// TIA Portal V17 export
// export: Created 2023-04-03T06:31:34.8487643Z, ExportSetting WithDefaults, DisplayName Totally Integrated Automation Portal, DisplayVersion V17 Update 4, DisplayName TIA Portal Openness, DisplayVersion V17 Update 4, DisplayName TIA Portal Version Control Interface, DisplayVersion V17, DisplayName STEP 7 Professional, DisplayVersion V17 Update 4, DisplayName STEP 7 Safety, DisplayVersion V17, DisplayName WinCC Professional, DisplayVersion V17 Update 4
FUNCTION "SM1_Logic" : Void   // FC60, LAD
TITLE = State Machine Logic
{ S7_Optimized_Access := 'TRUE' }
VERSION : 0.1
// stored: AutoNumber false, IsIECCheckEnabled false, SetENOAutomatically false, UDAEnableTagReadback false
   VAR_TEMP
      xStopSubSystem : Bool;
   END_VAR
   VAR_TEMP   // added for the SCL form of the ladder/FBD networks
      _w1 : Bool;
   END_VAR
BEGIN

REGION Network 1: Stop Command Local Mode
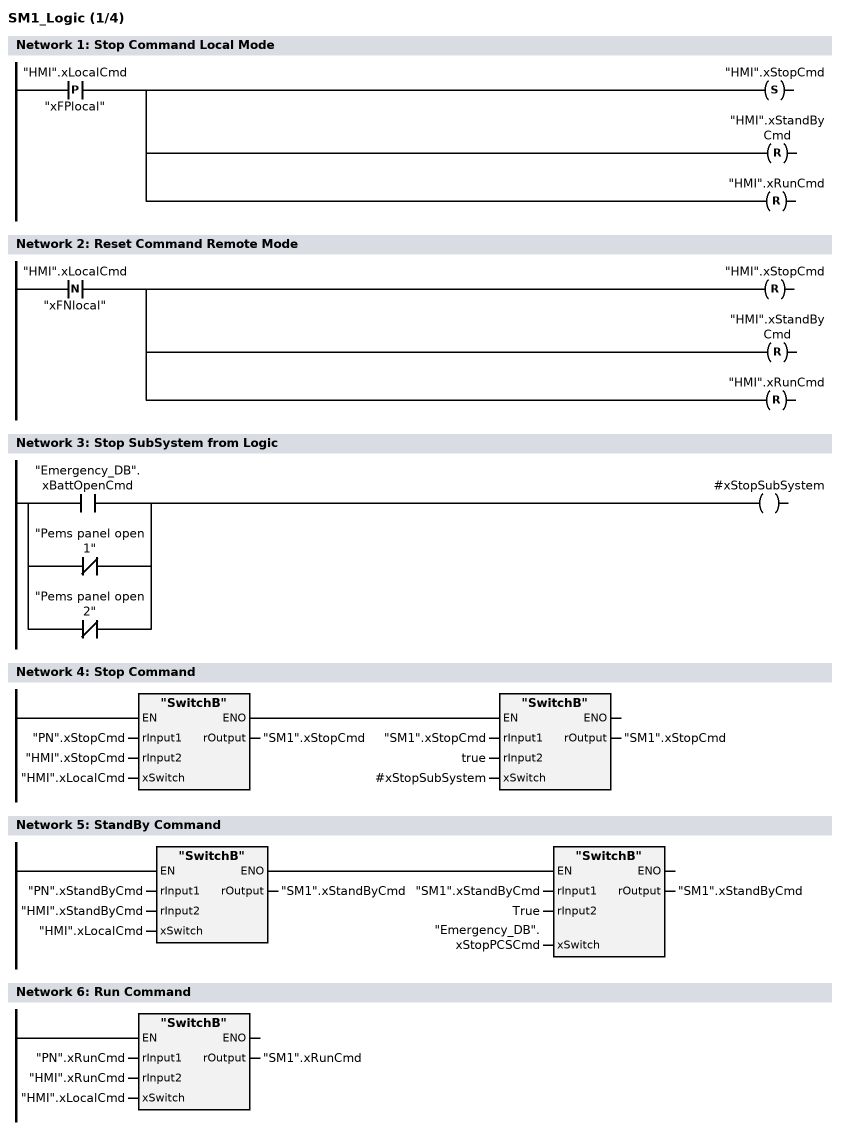
   RUNG wire#powerrail
      P_Contact(operand := "HMI".xLocalCmd, bit := "xFPlocal")
      wire#w1
      S_Coil( "HMI".xStopCmd )
   END_RUNG
   RUNG wire#w1
      R_Coil( "HMI".xStandByCmd )
   END_RUNG
   RUNG wire#w1
      R_Coil( "HMI".xRunCmd )
   END_RUNG
   // the same network as SCL:
   #_w1 := "HMI".xLocalCmd AND NOT "xFPlocal";   // rising edge of "HMI".xLocalCmd
   "xFPlocal" := "HMI".xLocalCmd;
   IF #_w1 THEN
       "HMI".xStopCmd := TRUE;
       "HMI".xStandByCmd := FALSE;
       "HMI".xRunCmd := FALSE;
   END_IF;
END_REGION

REGION Network 2: Reset Command Remote Mode
   RUNG wire#powerrail
      N_Contact(operand := "HMI".xLocalCmd, bit := "xFNlocal")
      wire#w1
      R_Coil( "HMI".xStopCmd )
   END_RUNG
   RUNG wire#w1
      R_Coil( "HMI".xStandByCmd )
   END_RUNG
   RUNG wire#w1
      R_Coil( "HMI".xRunCmd )
   END_RUNG
   // the same network as SCL:
   #_w1 := NOT "HMI".xLocalCmd AND "xFNlocal";   // falling edge of "HMI".xLocalCmd
   "xFNlocal" := "HMI".xLocalCmd;
   IF #_w1 THEN
       "HMI".xStopCmd := FALSE;
       "HMI".xStandByCmd := FALSE;
       "HMI".xRunCmd := FALSE;
   END_IF;
END_REGION

REGION Network 3: Stop SubSystem from Logic
   RUNG wire#powerrail
      Contact( "Emergency_DB".xBattOpenCmd )
      wire#w1
      Coil( #xStopSubSystem )
   END_RUNG
   RUNG wire#powerrail
      I_Contact( "Pems panel open 1" )
   END_RUNG wire#w1
   RUNG wire#powerrail
      I_Contact( "Pems panel open 2" )
   END_RUNG wire#w1
   // the same network as SCL:
   #xStopSubSystem := "Emergency_DB".xBattOpenCmd OR NOT "Pems panel open 1" OR NOT "Pems panel open 2";
END_REGION

REGION Network 4: Stop Command
   RUNG wire#powerrail
      "SwitchB"(rInput1 := "PN".xStopCmd, rInput2 := "HMI".xStopCmd, xSwitch := "HMI".xLocalCmd, rOutput => "SM1".xStopCmd)
      "SwitchB"(rInput1 := "SM1".xStopCmd, rInput2 := true, xSwitch := #xStopSubSystem, rOutput => "SM1".xStopCmd)
   END_RUNG
   // the same network as SCL:
   "SwitchB"(rInput1 := "PN".xStopCmd,
             rInput2 := "HMI".xStopCmd,
             xSwitch := "HMI".xLocalCmd,
             rOutput => "SM1".xStopCmd,
             ENO => #_w1);
   IF #_w1 THEN
       "SwitchB"(rInput1 := "SM1".xStopCmd, rInput2 := true, xSwitch := #xStopSubSystem, rOutput => "SM1".xStopCmd);
   END_IF;
END_REGION

REGION Network 5: StandBy Command
   RUNG wire#powerrail
      "SwitchB"(rInput1 := "PN".xStandByCmd, rInput2 := "HMI".xStandByCmd, xSwitch := "HMI".xLocalCmd, rOutput => "SM1".xStandByCmd)
      "SwitchB"(rInput1 := "SM1".xStandByCmd, rInput2 := True, xSwitch := "Emergency_DB".xStopPCSCmd, rOutput => "SM1".xStandByCmd)
   END_RUNG
   // the same network as SCL:
   "SwitchB"(rInput1 := "PN".xStandByCmd,
             rInput2 := "HMI".xStandByCmd,
             xSwitch := "HMI".xLocalCmd,
             rOutput => "SM1".xStandByCmd,
             ENO => #_w1);
   IF #_w1 THEN
       "SwitchB"(rInput1 := "SM1".xStandByCmd,
                 rInput2 := True,
                 xSwitch := "Emergency_DB".xStopPCSCmd,
                 rOutput => "SM1".xStandByCmd);
   END_IF;
END_REGION

REGION Network 6: Run Command
   RUNG wire#powerrail
      "SwitchB"(rInput1 := "PN".xRunCmd, rInput2 := "HMI".xRunCmd, xSwitch := "HMI".xLocalCmd, rOutput => "SM1".xRunCmd)
   END_RUNG
   // the same network as SCL:
   "SwitchB"(rInput1 := "PN".xRunCmd,
             rInput2 := "HMI".xRunCmd,
             xSwitch := "HMI".xLocalCmd,
             rOutput => "SM1".xRunCmd);
END_REGION

REGION Network 7: Local - Stop - StandBy - Run Status -> to HMI status
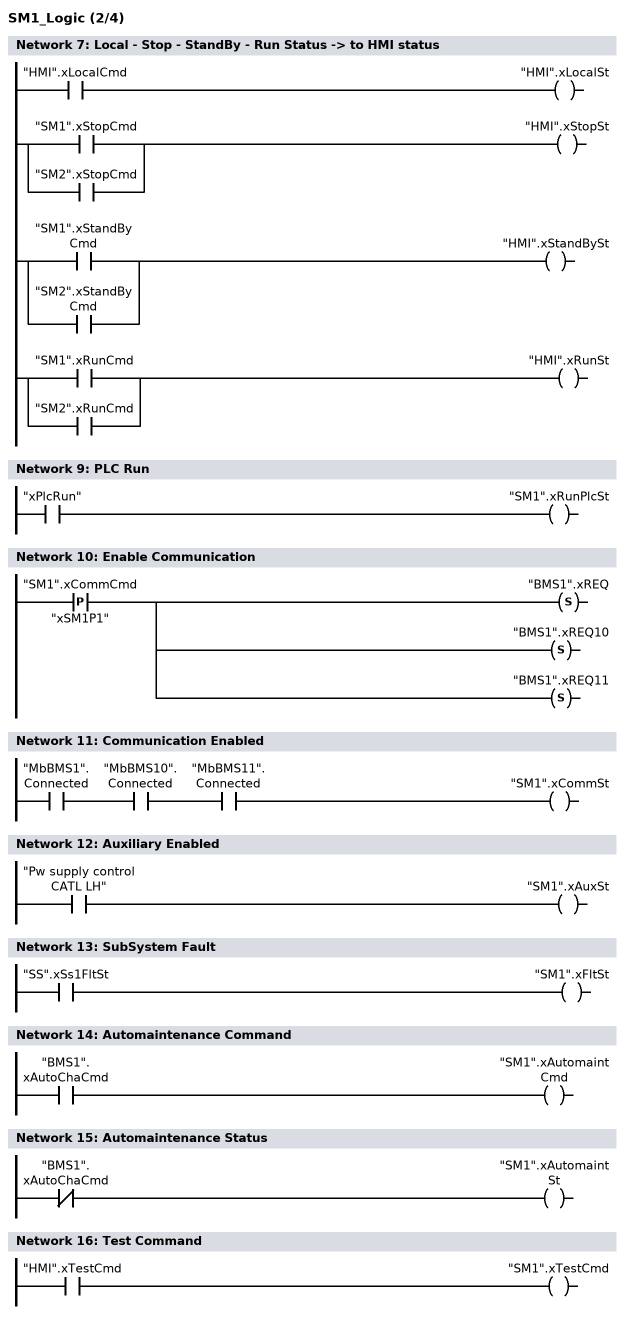
   RUNG wire#powerrail
      Contact( "HMI".xLocalCmd )
      Coil( "HMI".xLocalSt )
   END_RUNG
   RUNG wire#powerrail
      Contact( "SM1".xStopCmd )
      wire#w1
      Coil( "HMI".xStopSt )
   END_RUNG
   RUNG wire#powerrail
      Contact( "SM2".xStopCmd )
   END_RUNG wire#w1
   RUNG wire#powerrail
      Contact( "SM1".xStandByCmd )
      wire#w2
      Coil( "HMI".xStandBySt )
   END_RUNG
   RUNG wire#powerrail
      Contact( "SM2".xStandByCmd )
   END_RUNG wire#w2
   RUNG wire#powerrail
      Contact( "SM1".xRunCmd )
      wire#w3
      Coil( "HMI".xRunSt )
   END_RUNG
   RUNG wire#powerrail
      Contact( "SM2".xRunCmd )
   END_RUNG wire#w3
   // the same network as SCL:
   "HMI".xLocalSt := "HMI".xLocalCmd;
   "HMI".xStopSt := "SM1".xStopCmd OR "SM2".xStopCmd;
   "HMI".xStandBySt := "SM1".xStandByCmd OR "SM2".xStandByCmd;
   "HMI".xRunSt := "SM1".xRunCmd OR "SM2".xRunCmd;
END_REGION

REGION Network 9: PLC Run
   RUNG wire#powerrail
      Contact( "xPlcRun" )
      Coil( "SM1".xRunPlcSt )
   END_RUNG
   // the same network as SCL:
   "SM1".xRunPlcSt := "xPlcRun";
END_REGION

REGION Network 10: Enable Communication
   RUNG wire#powerrail
      P_Contact(operand := "SM1".xCommCmd, bit := "xSM1P1")
      wire#w1
      S_Coil( "BMS1".xREQ )
   END_RUNG
   RUNG wire#w1
      S_Coil( "BMS1".xREQ10 )
   END_RUNG
   RUNG wire#w1
      S_Coil( "BMS1".xREQ11 )
   END_RUNG
   // the same network as SCL:
   #_w1 := "SM1".xCommCmd AND NOT "xSM1P1";   // rising edge of "SM1".xCommCmd
   "xSM1P1" := "SM1".xCommCmd;
   IF #_w1 THEN
       "BMS1".xREQ := TRUE;
       "BMS1".xREQ10 := TRUE;
       "BMS1".xREQ11 := TRUE;
   END_IF;
END_REGION

REGION Network 11: Communication Enabled
   RUNG wire#powerrail
      Contact( "MbBMS1".Connected )
      Contact( "MbBMS10".Connected )
      Contact( "MbBMS11".Connected )
      Coil( "SM1".xCommSt )
   END_RUNG
   // the same network as SCL:
   "SM1".xCommSt := "MbBMS1".Connected AND "MbBMS10".Connected AND "MbBMS11".Connected;
END_REGION

REGION Network 12: Auxiliary Enabled
   RUNG wire#powerrail
      Contact( "Pw supply control CATL LH" )
      Coil( "SM1".xAuxSt )
   END_RUNG
   // the same network as SCL:
   "SM1".xAuxSt := "Pw supply control CATL LH";
END_REGION

REGION Network 13: SubSystem Fault
   RUNG wire#powerrail
      Contact( "SS".xSs1FltSt )
      Coil( "SM1".xFltSt )
   END_RUNG
   // the same network as SCL:
   "SM1".xFltSt := "SS".xSs1FltSt;
END_REGION

REGION Network 14: Automaintenance Command
   RUNG wire#powerrail
      Contact( "BMS1".xAutoChaCmd )
      Coil( "SM1".xAutomaintCmd )
   END_RUNG
   // the same network as SCL:
   "SM1".xAutomaintCmd := "BMS1".xAutoChaCmd;
END_REGION

REGION Network 15: Automaintenance Status
   RUNG wire#powerrail
      I_Contact( "BMS1".xAutoChaCmd )
      Coil( "SM1".xAutomaintSt )
   END_RUNG
   // the same network as SCL:
   "SM1".xAutomaintSt := NOT "BMS1".xAutoChaCmd;
END_REGION

REGION Network 16: Test Command
   RUNG wire#powerrail
      Contact( "HMI".xTestCmd )
      Coil( "SM1".xTestCmd )
   END_RUNG
   // the same network as SCL:
   "SM1".xTestCmd := "HMI".xTestCmd;
END_REGION

REGION Network 17: Ready condition on the Power Island - to check
   // - primo contatto era "MV ok" from PN 
   // -gli altri sono i DC breaker close dei PE
   // -e un bypass icoming UPS line from grid
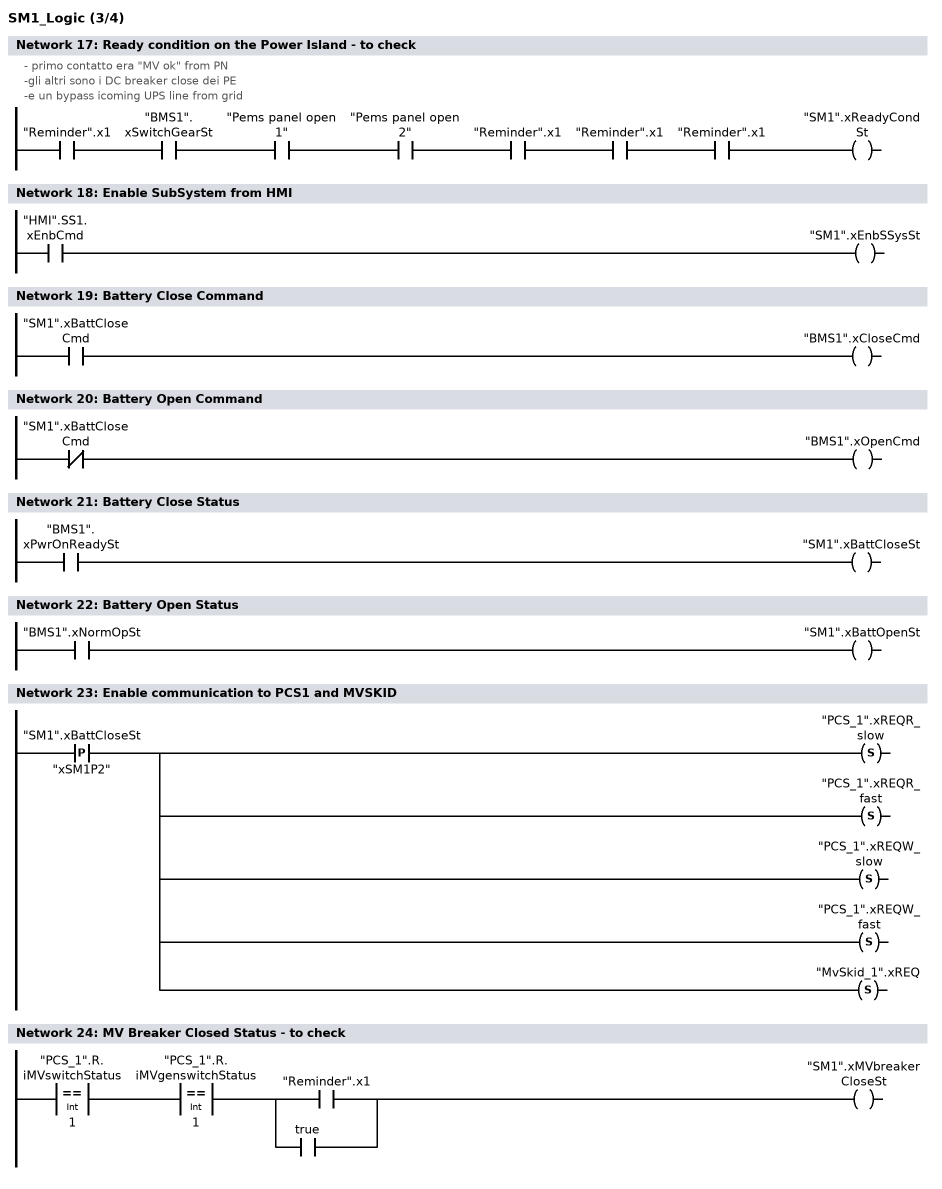
   RUNG wire#powerrail
      Contact( "Reminder".x1 )
      Contact( "BMS1".xSwitchGearSt )
      Contact( "Pems panel open 1" )
      Contact( "Pems panel open 2" )
      Contact( "Reminder".x1 )
      Contact( "Reminder".x1 )
      Contact( "Reminder".x1 )
      Coil( "SM1".xReadyCondSt )
   END_RUNG
   // the same network as SCL:
   "SM1".xReadyCondSt := "Reminder".x1 AND "BMS1".xSwitchGearSt AND "Pems panel open 1" AND "Pems panel open 2" AND "Reminder".x1 AND "Reminder".x1 AND "Reminder".x1;
END_REGION

REGION Network 18: Enable SubSystem from HMI
   RUNG wire#powerrail
      Contact( "HMI".SS1.xEnbCmd )
      Coil( "SM1".xEnbSSysSt )
   END_RUNG
   // the same network as SCL:
   "SM1".xEnbSSysSt := "HMI".SS1.xEnbCmd;
END_REGION

REGION Network 19: Battery Close Command
   RUNG wire#powerrail
      Contact( "SM1".xBattCloseCmd )
      Coil( "BMS1".xCloseCmd )
   END_RUNG
   // the same network as SCL:
   "BMS1".xCloseCmd := "SM1".xBattCloseCmd;
END_REGION

REGION Network 20: Battery Open Command
   RUNG wire#powerrail
      I_Contact( "SM1".xBattCloseCmd )
      Coil( "BMS1".xOpenCmd )
   END_RUNG
   // the same network as SCL:
   "BMS1".xOpenCmd := NOT "SM1".xBattCloseCmd;
END_REGION

REGION Network 21: Battery Close Status
   RUNG wire#powerrail
      Contact( "BMS1".xPwrOnReadySt )
      Coil( "SM1".xBattCloseSt )
   END_RUNG
   // the same network as SCL:
   "SM1".xBattCloseSt := "BMS1".xPwrOnReadySt;
END_REGION

REGION Network 22: Battery Open Status
   RUNG wire#powerrail
      Contact( "BMS1".xNormOpSt )
      Coil( "SM1".xBattOpenSt )
   END_RUNG
   // the same network as SCL:
   "SM1".xBattOpenSt := "BMS1".xNormOpSt;
END_REGION

REGION Network 23: Enable communication to PCS1 and MVSKID
   RUNG wire#powerrail
      P_Contact(operand := "SM1".xBattCloseSt, bit := "xSM1P2")
      wire#w1
      S_Coil( "PCS_1".xREQR_slow )
   END_RUNG
   RUNG wire#w1
      S_Coil( "PCS_1".xREQR_fast )
   END_RUNG
   RUNG wire#w1
      S_Coil( "PCS_1".xREQW_slow )
   END_RUNG
   RUNG wire#w1
      S_Coil( "PCS_1".xREQW_fast )
   END_RUNG
   RUNG wire#w1
      S_Coil( "MvSkid_1".xREQ )
   END_RUNG
   // the same network as SCL:
   #_w1 := "SM1".xBattCloseSt AND NOT "xSM1P2";   // rising edge of "SM1".xBattCloseSt
   "xSM1P2" := "SM1".xBattCloseSt;
   IF #_w1 THEN
       "PCS_1".xREQR_slow := TRUE;
       "PCS_1".xREQR_fast := TRUE;
       "PCS_1".xREQW_slow := TRUE;
       "PCS_1".xREQW_fast := TRUE;
       "MvSkid_1".xREQ := TRUE;
   END_IF;
END_REGION

REGION Network 24: MV Breaker Closed Status - to check
   RUNG wire#powerrail
      { S7_Templates := "SrcType := Int" } EQ_Contact(in1 := "PCS_1".R.iMVswitchStatus, in2 := 1)
      { S7_Templates := "SrcType := Int" } EQ_Contact(in1 := "PCS_1".R.iMVgenswitchStatus, in2 := 1)
      wire#w1
      Contact( "Reminder".x1 )
      wire#w2
      Coil( "SM1".xMVbreakerCloseSt )
   END_RUNG
   RUNG wire#w1
      Contact( true )
   END_RUNG wire#w2
   // the same network as SCL:
   "SM1".xMVbreakerCloseSt := ("PCS_1".R.iMVswitchStatus = 1) AND ("PCS_1".R.iMVgenswitchStatus = 1) AND ("Reminder".x1 OR true);
END_REGION

REGION Network 25: MV Breaker Open Status
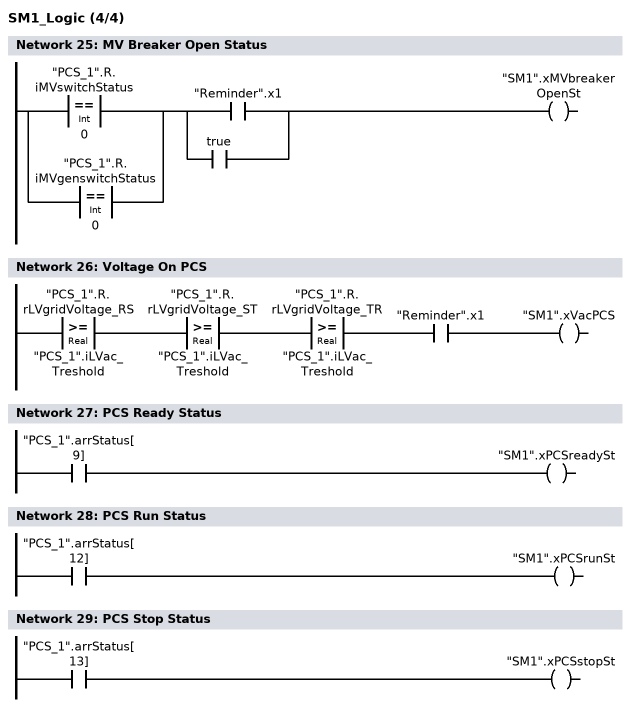
   RUNG wire#powerrail
      { S7_Templates := "SrcType := Int" } EQ_Contact(in1 := "PCS_1".R.iMVswitchStatus, in2 := 0)
      wire#w1
      Contact( "Reminder".x1 )
      wire#w2
      Coil( "SM1".xMVbreakerOpenSt )
   END_RUNG
   RUNG wire#powerrail
      { S7_Templates := "SrcType := Int" } EQ_Contact(in1 := "PCS_1".R.iMVgenswitchStatus, in2 := 0)
   END_RUNG wire#w1
   RUNG wire#w1
      Contact( true )
   END_RUNG wire#w2
   // the same network as SCL:
   "SM1".xMVbreakerOpenSt := (("PCS_1".R.iMVswitchStatus = 0) OR ("PCS_1".R.iMVgenswitchStatus = 0)) AND ("Reminder".x1 OR true);
END_REGION

REGION Network 26: Voltage On PCS
   RUNG wire#powerrail
      { S7_Templates := "SrcType := Real" } GE_Contact(in1 := "PCS_1".R.rLVgridVoltage_RS, in2 := "PCS_1".iLVac_Treshold)
      { S7_Templates := "SrcType := Real" } GE_Contact(in1 := "PCS_1".R.rLVgridVoltage_ST, in2 := "PCS_1".iLVac_Treshold)
      { S7_Templates := "SrcType := Real" } GE_Contact(in1 := "PCS_1".R.rLVgridVoltage_TR, in2 := "PCS_1".iLVac_Treshold)
      Contact( "Reminder".x1 )
      Coil( "SM1".xVacPCS )
   END_RUNG
   // the same network as SCL:
   "SM1".xVacPCS := ("PCS_1".R.rLVgridVoltage_RS >= "PCS_1".iLVac_Treshold) AND ("PCS_1".R.rLVgridVoltage_ST >= "PCS_1".iLVac_Treshold) AND ("PCS_1".R.rLVgridVoltage_TR >= "PCS_1".iLVac_Treshold) AND "Reminder".x1;
END_REGION

REGION Network 27: PCS Ready Status
   RUNG wire#powerrail
      Contact( "PCS_1".arrStatus[9] )
      Coil( "SM1".xPCSreadySt )
   END_RUNG
   // the same network as SCL:
   "SM1".xPCSreadySt := "PCS_1".arrStatus[9];
END_REGION

REGION Network 28: PCS Run Status
   RUNG wire#powerrail
      Contact( "PCS_1".arrStatus[12] )
      Coil( "SM1".xPCSrunSt )
   END_RUNG
   // the same network as SCL:
   "SM1".xPCSrunSt := "PCS_1".arrStatus[12];
END_REGION

REGION Network 29: PCS Stop Status
   RUNG wire#powerrail
      Contact( "PCS_1".arrStatus[13] )
      Coil( "SM1".xPCSstopSt )
   END_RUNG
   // the same network as SCL:
   "SM1".xPCSstopSt := "PCS_1".arrStatus[13];
END_REGION
END_FUNCTION
